# EPICS IOC start-up script: iocsh/ethercatmcLongoutReadback.iocsh
ethercatmcCreateAsynParam $(MOTOR_PORT) $(ASYNPARAMNAME) Int32

dbLoadRecords("ethercatmcLongoutReadback.template", "P=$(P), R=$(R), MOTOR_PORT=$(MOTOR_PORT), ASYNPARAMNAME=$(ASYNPARAMNAME), CHNO=$(CHNO=0), DESC=$(DESC), EGU=$(EGU) ")
